PROGRAM WatchDog_PLC
VAR
	TON_0: TON;
END_VAR

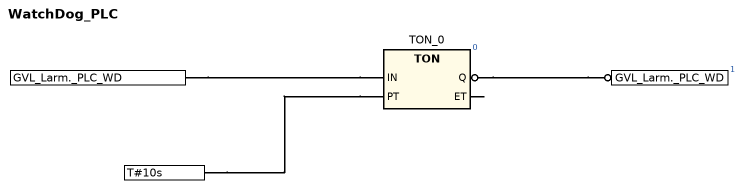
TON_0(IN := GVL_Larm._PLC_WD, PT := T#10s); // TON
GVL_Larm._PLC_WD := NOT (NOT TON_0.Q);

END_PROGRAM

(* stored: Version 1.1.0.1, ProductVersion 3.1.4020.12
   POU WatchDog_PLC: Id {7f935a52-0c74-47cf-bde9-ff29b6126410}, SpecialFunc None *)
